{attribute addProperty BoxType "EP9214-0023-0019"}
{attribute addProperty Id "Enable_Control_Via_FieldbusAT %Q*BOOL811Global_ResetAT %Q*BOOL814"}
{attribute addProperty CRC "1857578072"}
{attribute addProperty SizeInBites "16"}
{attribute addProperty SizeInBytes "2"}
TYPE DPO_Outputs_Device_6EB86458 :
STRUCT
	{attribute addProperty Name "Enable_Control_Via_Fieldbus"}
	Enable_Control_Via_Fieldbus AT %Q* : BOOL;
	{attribute addProperty Name "Global_Reset"}
	Global_Reset AT %Q* : BOOL;
END_STRUCT
END_TYPE

(* stored: Version 1.2.0.0, ProductVersion 3.1.4024.9
   DUT DPO_Outputs_Device_6EB86458: Id {e9e463c5-51b6-4d81-a7e6-3212b65fb87a} *)
